INTERFACE I_STREAM

PROPERTY BufferSize : UDINT
GET
END_GET
END_PROPERTY

METHOD Close : DINT
VAR_INPUT
END_VAR
END_METHOD

PROPERTY EndOfStream : BOOL
GET
END_GET
END_PROPERTY

PROPERTY IsValid : BOOL
GET
END_GET
END_PROPERTY

METHOD Peek : DINT
VAR_INPUT
	ptr_DataOut : POINTER TO BYTE;
END_VAR
END_METHOD

PROPERTY Position : UDINT
GET
END_GET
END_PROPERTY

METHOD Read : DINT
VAR_INPUT
	ptr_DataOut : PVOID;
	Length		: UDINT;
END_VAR
END_METHOD

METHOD Seek : DINT
VAR_INPUT
	Offset 		: UDINT;
	SeekStyle 	: E_STREAMSEEKTYPE;
END_VAR
END_METHOD

METHOD Write : DINT
VAR_INPUT
	ptr_DataIn	: PVOID;
	Length		: UDINT;
END_VAR
END_METHOD

END_INTERFACE

(* stored: Version 1.1.0.1, ProductVersion 3.1.4020.3
   Itf I_STREAM: Id {5953bfdd-a48b-492a-8c79-c85297f262b9}
   Folder Methods: Id {56776e1f-2871-4f00-b8cd-81b909631ce0}
   Folder Properties: Id {ce63abcd-9d4d-4c5d-bee2-b335a96933fc}
   Property BufferSize: Id {c34623ff-2a57-426e-9040-e574610d22c1}
   Get Get: Id {7b4c4e1e-56d7-4a56-a628-da38827bbb2e}
   Method Close: Id {bff1604a-fcb7-4ff1-b43a-637de2b8f049}
   Property EndOfStream: Id {a2d4d65e-a939-4187-8b6b-aa87b84d2607}
   Get Get: Id {1aad2dfb-9cba-4b96-9d3e-9bc2a19318b2}
   Property IsValid: Id {ac69761a-0435-4af0-bd1f-5705d786d8a1}
   Get Get: Id {0903634d-092e-4a4b-8715-b863d40231f0}
   Method Peek: Id {045b16e8-4d45-45b7-baf5-0fa9c4b7503c}
   Property Position: Id {715bd596-28d4-44c9-aaec-3c9a90d6dfab}
   Get Get: Id {e179f4bd-a493-4d3f-89f8-b7f480327d3b}
   Method Read: Id {47521f98-ffb6-4e89-a486-d3df4188fd2c}
   Method Seek: Id {a9835b55-ed84-4d8c-857e-520d4704ffd4}
   Method Write: Id {15d84086-0ea3-4075-a1ad-afdb7c819e01} *)
